FUNCTION F_STRING_TO_ARG : T_Arg
VAR_IN_OUT
    in : T_MaxString;
END_VAR
VAR
    Result : T_Arg;
END_VAR

Result.eType := E_ArgType.ARGTYPE_STRING;
Result.pData := ADR(in);
Result.cbLen := SIZEOF(in); // not LEN()! F_STRING gives LEN which does not work with CallRPC_Method args!

F_STRING_TO_ARG := Result;

END_FUNCTION

(* stored: Version 1.1.0.1, ProductVersion 3.1.4024.3
   POU F_STRING_TO_ARG: Id {c7852143-9abe-0d35-20ea-eebcd7c9f5ff}, SpecialFunc None *)
